PROGRAM MAIN
VAR
	AutomationRunner : SignalControlledIntersectionAutomationRunner;
END_VAR

AutomationRunner.Run();

END_PROGRAM

(* stored: Version 1.1.0.1
   POU MAIN: Id {ca65afb8-727d-41a0-9d5d-3e437a913e63}, SpecialFunc None *)
